TYPE CmpCore :
STRUCT
	
	Framework: Framework;

END_STRUCT
END_TYPE

(* stored: Version 1.1.0.1, ProductVersion 3.1.4024.6
   DUT CmpCore: Id {e0c673d6-c696-47f3-9bb8-4807b7df0cf4} *)
